TYPE T_Ctrl_SIf_PCE_Cfg :
STRUCT
END_STRUCT
END_TYPE

(* stored: Version 1.1.0.1, ProductVersion 3.1.0.19
   DUT T_Ctrl_SIf_PCE_Cfg: Id {914dc26f-68b7-4b49-9271-71c3e42a4ebf} *)
